// TIA Portal V20 export
// export: Created 2026-07-16T12:58:51.2791599Z, ExportSetting WithDefaults, DisplayName Totally Integrated Automation Portal, DisplayVersion V20 Update 5, DisplayName TIA Portal Openness, DisplayVersion V20 Update 4, DisplayName TIA Portal Version Control Interface, DisplayVersion V20 Update 5, DisplayName SINAMICS Startdrive Advanced, DisplayVersion V20, DisplayName SINAMICS DCC, DisplayVersion V20, DisplayName SINAMICS Startdrive G130, G150, S120, S150, SINAMICS MV, G220, S200, S210, DisplayVersion V20, DisplayName SINAMICS Startdrive G110M, G120, G120C, G120D, G120P, G115D, DisplayVersion V20, DisplayName STEP 7 Professional, DisplayVersion V20 Update 5, DisplayName STEP 7 Safety, DisplayVersion V20 Update 2, DisplayName WinCC Basic/Comfort/Advanced, DisplayVersion V20 Update 5, DisplayName WinCC Unified, DisplayVersion V20 Update 5
FUNCTION_BLOCK "FB_PusherControl"   // FB3, LAD
TITLE = Pusher Control
{ S7_Optimized_Access := 'TRUE' }
VERSION : 0.1
// Pusher ram sequencing (C-118-C-125). Step legend (C-120): 0=Parked (idle/home, ram fully retracted, no motion) - 10=DriveToEndTravel (forward stroke in progress) - 20=Hold (paused at full travel, brief settle before retracting) - 30=Retract (returning to home; also the recovery/abort target from any bad state). Mode legend: 0=Off (finish a retract already in progress, then park; no new cycle starts) - 1=Auto (hopper-high-level starts a cycle) - 2=Manual (operator button/jog starts a cycle).
// stored: AutoNumber true, IsIECCheckEnabled false, IsRetainMemResEnabled false, MemoryReserve 100, SetENOAutomatically false, UDAEnableTagReadback false
   VAR RETAIN
      IO { S7_SetPoint := 'True'} : "UDT_PusherIO";   // Caller-visible interface (C-115) - FC_ControlMain writes Mode/HopperHighLevel/limits/tunables in, reads Extend/Retract/RunPowerPack/fault bits out. See the block header for the Step/Mode value legend.
   END_VAR
   VAR
      EndTravelTimeoutMS : DInt;
      ParkedTimeoutMS : DInt;
      EndTravelHoldTimeMS : DInt;
      PumpRunOnTimeMS : DInt;
      JogWarningTimeMS : DInt;
      PressureTripConfirmTimeMS : DInt;
      PressureClearResumeDelayMS : DInt;
      PressureConfirmTimer { S7_SetPoint := 'True'} : TON_TIME;
      PressureClearTimer { S7_SetPoint := 'True'} : TON_TIME;
      PressureHold : Bool;   // Latched jam hold, not a fault (C-123) - see the Pressure Detection network. Freezes ExtendDemand while set; clears itself once pressure has genuinely stayed clear for PressureClearResumeDelay.
      PressureConfirmEdge : Bool;
      PressureConfirmEdgeMem : Bool;
      PressureTripCount : Int;   // Confirmed jams this cycle - reset each cycle start, not time-windowed. Compared against IO.PressureTripCountThreshold to raise Blocked.
      EndTravelTimer { S7_SetPoint := 'True'} : TON_TIME;
      HoldTimer { S7_SetPoint := 'True'} : TON_TIME;
      ParkedTimer { S7_SetPoint := 'True'} : TON_TIME;
      JogPreStartTimer { S7_SetPoint := 'True'} : TON_TIME;
      ExtendDemand : Bool;
      RetractDemand : Bool;
      PumpDemand : Bool;   // ExtendDemand OR RetractDemand - the pump's own immediate (non-run-on) demand signal.
      PumpEverDemanded : Bool;   // Cold-start guard for the pump run-on off-delay below - see that network's own comment.
      PumpRunOnTimer { S7_SetPoint := 'True'} : TON_TIME;
   END_VAR
   VAR_TEMP
      "Time" : Real;
   END_VAR
BEGIN

REGION Network 1: Enable
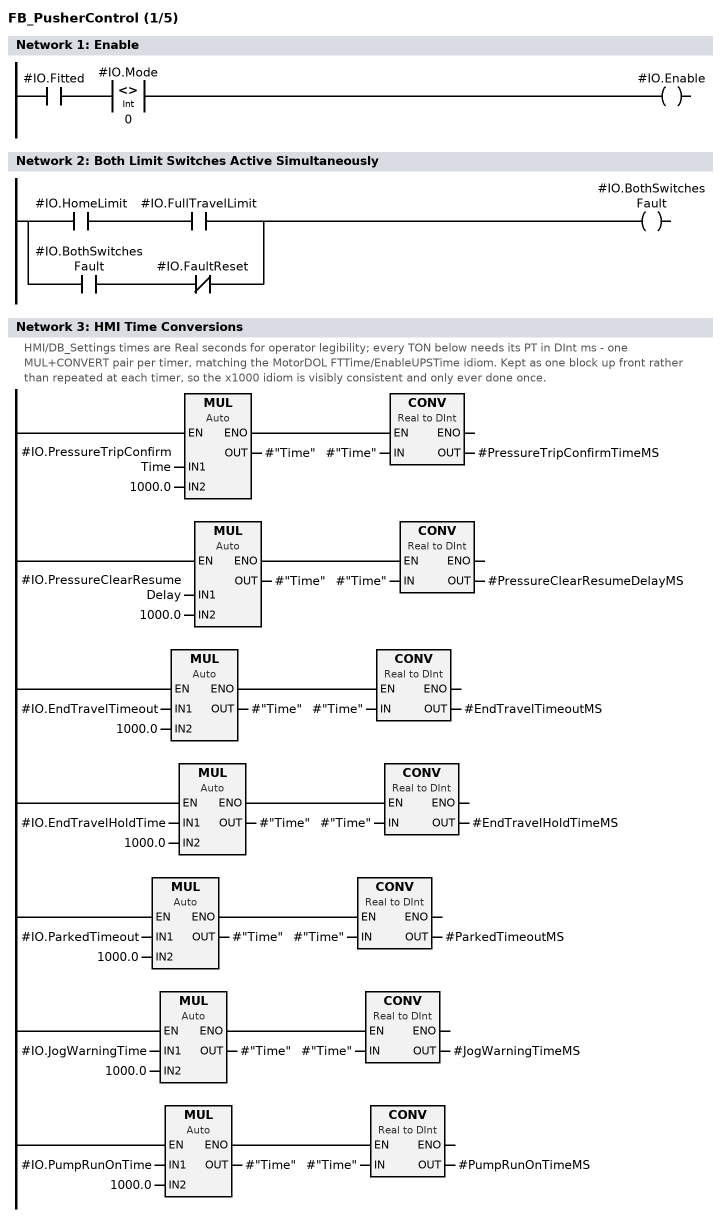
   RUNG wire#powerrail
      Contact( #IO.Fitted )
      { S7_Templates := "SrcType := Int" } NE_Contact(in1 := #IO.Mode, in2 := 0)
      Coil( #IO.Enable )
   END_RUNG
   // the same network as SCL:
   #IO.Enable := #IO.Fitted AND (#IO.Mode <> 0);
END_REGION

REGION Network 2: Both Limit Switches Active Simultaneously
   RUNG wire#powerrail
      Contact( #IO.HomeLimit )
      Contact( #IO.FullTravelLimit )
      wire#w1
      Coil( #IO.BothSwitchesFault )
   END_RUNG
   RUNG wire#powerrail
      Contact( #IO.BothSwitchesFault )
      I_Contact( #IO.FaultReset )
   END_RUNG wire#w1
   // the same network as SCL:
   #IO.BothSwitchesFault := (#IO.HomeLimit AND #IO.FullTravelLimit) OR (#IO.BothSwitchesFault AND NOT #IO.FaultReset);
END_REGION

REGION Network 3: HMI Time Conversions
   // HMI/DB_Settings times are Real seconds for operator legibility; every TON below needs its PT in DInt ms - one MUL+CONVERT pair per timer, matching the MotorDOL FTTime/EnableUPSTime idiom. Kept as one block up front rather than repeated at each timer, so the x1000 idiom is visibly consistent and only ever done once.
   RUNG wire#powerrail
      Mul(in1 := #IO.PressureTripConfirmTime, in2 := 1000.0, out => #"Time")
      { S7_Templates := "[SrcType := Real, DestType := DInt]" } Convert(in := #"Time", out => #PressureTripConfirmTimeMS)
   END_RUNG
   RUNG wire#powerrail
      Mul(in1 := #IO.PressureClearResumeDelay, in2 := 1000.0, out => #"Time")
      { S7_Templates := "[SrcType := Real, DestType := DInt]" } Convert(in := #"Time", out => #PressureClearResumeDelayMS)
   END_RUNG
   RUNG wire#powerrail
      Mul(in1 := #IO.EndTravelTimeout, in2 := 1000.0, out => #"Time")
      { S7_Templates := "[SrcType := Real, DestType := DInt]" } Convert(in := #"Time", out => #EndTravelTimeoutMS)
   END_RUNG
   RUNG wire#powerrail
      Mul(in1 := #IO.EndTravelHoldTime, in2 := 1000.0, out => #"Time")
      { S7_Templates := "[SrcType := Real, DestType := DInt]" } Convert(in := #"Time", out => #EndTravelHoldTimeMS)
   END_RUNG
   RUNG wire#powerrail
      Mul(in1 := #IO.ParkedTimeout, in2 := 1000.0, out => #"Time")
      { S7_Templates := "[SrcType := Real, DestType := DInt]" } Convert(in := #"Time", out => #ParkedTimeoutMS)
   END_RUNG
   RUNG wire#powerrail
      Mul(in1 := #IO.JogWarningTime, in2 := 1000.0, out => #"Time")
      { S7_Templates := "[SrcType := Real, DestType := DInt]" } Convert(in := #"Time", out => #JogWarningTimeMS)
   END_RUNG
   RUNG wire#powerrail
      Mul(in1 := #IO.PumpRunOnTime, in2 := 1000.0, out => #"Time")
      { S7_Templates := "[SrcType := Real, DestType := DInt]" } Convert(in := #"Time", out => #PumpRunOnTimeMS)
   END_RUNG
   // the same network as SCL:
   #"Time" := #IO.PressureTripConfirmTime * 1000.0;
   #PressureTripConfirmTimeMS := REAL_TO_DINT(#"Time");
   #"Time" := #IO.PressureClearResumeDelay * 1000.0;
   #PressureClearResumeDelayMS := REAL_TO_DINT(#"Time");
   #"Time" := #IO.EndTravelTimeout * 1000.0;
   #EndTravelTimeoutMS := REAL_TO_DINT(#"Time");
   #"Time" := #IO.EndTravelHoldTime * 1000.0;
   #EndTravelHoldTimeMS := REAL_TO_DINT(#"Time");
   #"Time" := #IO.ParkedTimeout * 1000.0;
   #ParkedTimeoutMS := REAL_TO_DINT(#"Time");
   #"Time" := #IO.JogWarningTime * 1000.0;
   #JogWarningTimeMS := REAL_TO_DINT(#"Time");
   #"Time" := #IO.PumpRunOnTime * 1000.0;
   #PumpRunOnTimeMS := REAL_TO_DINT(#"Time");
END_REGION

REGION Network 4: Pressure Trip Detection, Hold, And Counting
   // One function, one network: a trip must be debounced (PressureConfirmTimer) before it counts - momentary pressure spikes aren't a real jam. Hold latches through a confirmed trip and only releases once pressure has genuinely cleared for PressureClearResumeDelay, so a bouncing switch can't re-trigger the count on every scan. Count resets each cycle start (Step 0-to-10 launch condition), not on a rolling time window.
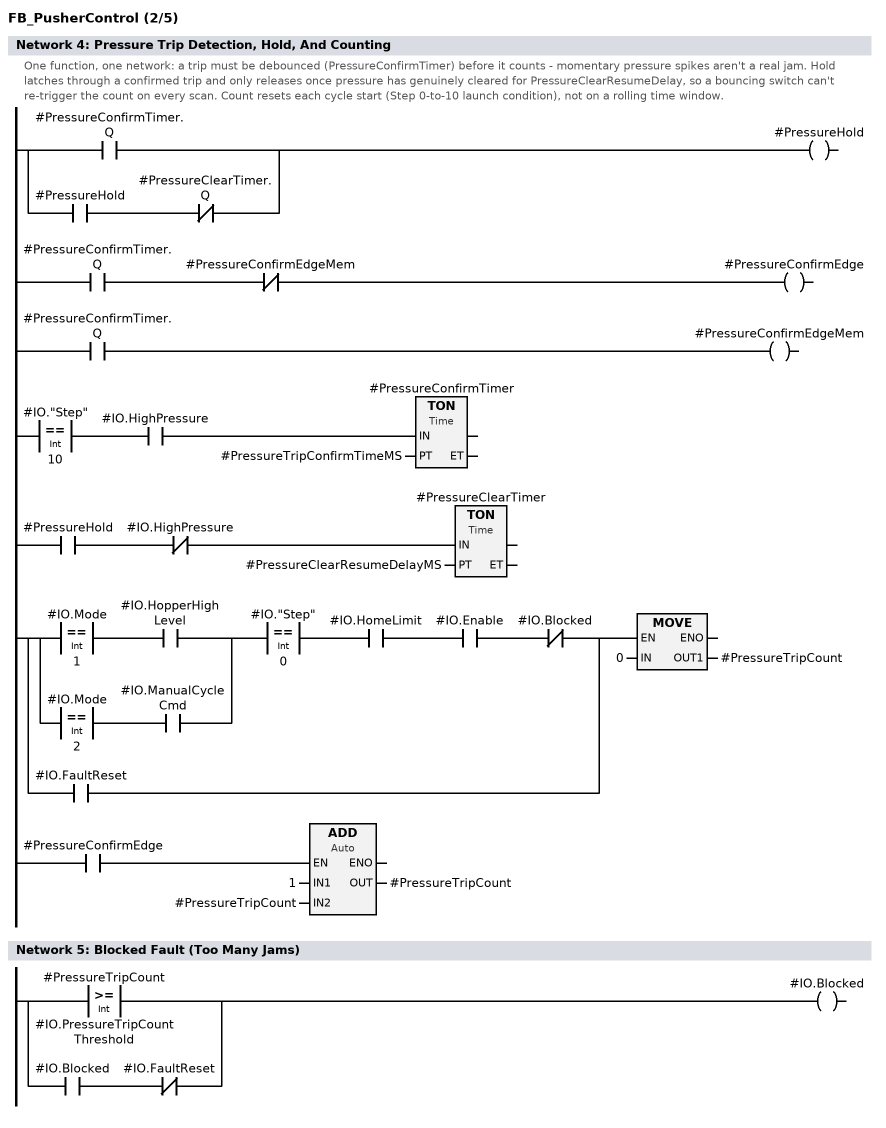
   RUNG wire#powerrail
      Contact( #PressureConfirmTimer.Q )
      wire#w1
      Coil( #PressureHold )
   END_RUNG
   RUNG wire#powerrail
      Contact( #PressureHold )
      I_Contact( #PressureClearTimer.Q )
   END_RUNG wire#w1
   RUNG wire#powerrail
      Contact( #PressureConfirmTimer.Q )
      I_Contact( #PressureConfirmEdgeMem )
      Coil( #PressureConfirmEdge )
   END_RUNG
   RUNG wire#powerrail
      Contact( #PressureConfirmTimer.Q )
      Coil( #PressureConfirmEdgeMem )
   END_RUNG
   RUNG wire#powerrail
      { S7_Templates := "SrcType := Int" } EQ_Contact(in1 := #IO."Step", in2 := 10)
      Contact( #IO.HighPressure )
      { S7_Templates := "time_type := Time" } #PressureConfirmTimer.TON(pt := #PressureTripConfirmTimeMS, et =>)
   END_RUNG
   RUNG wire#powerrail
      Contact( #PressureHold )
      I_Contact( #IO.HighPressure )
      { S7_Templates := "time_type := Time" } #PressureClearTimer.TON(pt := #PressureClearResumeDelayMS, et =>)
   END_RUNG
   RUNG wire#powerrail
      { S7_Templates := "SrcType := Int" } EQ_Contact(in1 := #IO.Mode, in2 := 1)
      Contact( #IO.HopperHighLevel )
      wire#w2
      { S7_Templates := "SrcType := Int" } EQ_Contact(in1 := #IO."Step", in2 := 0)
      Contact( #IO.HomeLimit )
      Contact( #IO.Enable )
      I_Contact( #IO.Blocked )
      wire#w3
      Move(in := 0, out1 => #PressureTripCount)
   END_RUNG
   RUNG wire#powerrail
      { S7_Templates := "SrcType := Int" } EQ_Contact(in1 := #IO.Mode, in2 := 2)
      Contact( #IO.ManualCycleCmd )
   END_RUNG wire#w2
   RUNG wire#powerrail
      Contact( #IO.FaultReset )
   END_RUNG wire#w3
   RUNG wire#powerrail
      Contact( #PressureConfirmEdge )
      Add(in1 := 1, in2 := #PressureTripCount, out => #PressureTripCount)
   END_RUNG
   // the same network as SCL:
   #PressureHold := #PressureConfirmTimer.Q OR (#PressureHold AND NOT #PressureClearTimer.Q);
   #PressureConfirmEdge := #PressureConfirmTimer.Q AND NOT #PressureConfirmEdgeMem;
   #PressureConfirmEdgeMem := #PressureConfirmTimer.Q;
   #PressureConfirmTimer(IN := (#IO."Step" = 10) AND #IO.HighPressure, PT := #PressureTripConfirmTimeMS);   // TON
   #PressureClearTimer(IN := #PressureHold AND NOT #IO.HighPressure, PT := #PressureClearResumeDelayMS);   // TON
   IF ((((#IO.Mode = 1) AND #IO.HopperHighLevel) OR ((#IO.Mode = 2) AND #IO.ManualCycleCmd)) AND (#IO."Step" = 0) AND #IO.HomeLimit AND #IO.Enable AND NOT #IO.Blocked) OR #IO.FaultReset THEN
       #PressureTripCount := 0;
   END_IF;
   IF #PressureConfirmEdge THEN #PressureTripCount := 1 + #PressureTripCount; END_IF;
END_REGION

REGION Network 5: Blocked Fault (Too Many Jams)
   RUNG wire#powerrail
      { S7_Templates := "SrcType := Int" } GE_Contact(in1 := #PressureTripCount, in2 := #IO.PressureTripCountThreshold)
      wire#w1
      Coil( #IO.Blocked )
   END_RUNG
   RUNG wire#powerrail
      Contact( #IO.Blocked )
      I_Contact( #IO.FaultReset )
   END_RUNG wire#w1
   // the same network as SCL:
   #IO.Blocked := (#PressureTripCount >= #IO.PressureTripCountThreshold) OR (#IO.Blocked AND NOT #IO.FaultReset);
END_REGION

REGION Network 6: Step 0 (Parked) - Transitions
   // Not-at-home while idle (power-up mid-stroke, or a cycle that ended without reaching HomeLimit) drives straight to Retract (30) to re-establish home before any new cycle is accepted - never straight back into a forward stroke from an unknown position. Suppressed during an active jog command so jogging isn't fought by an auto-retract.
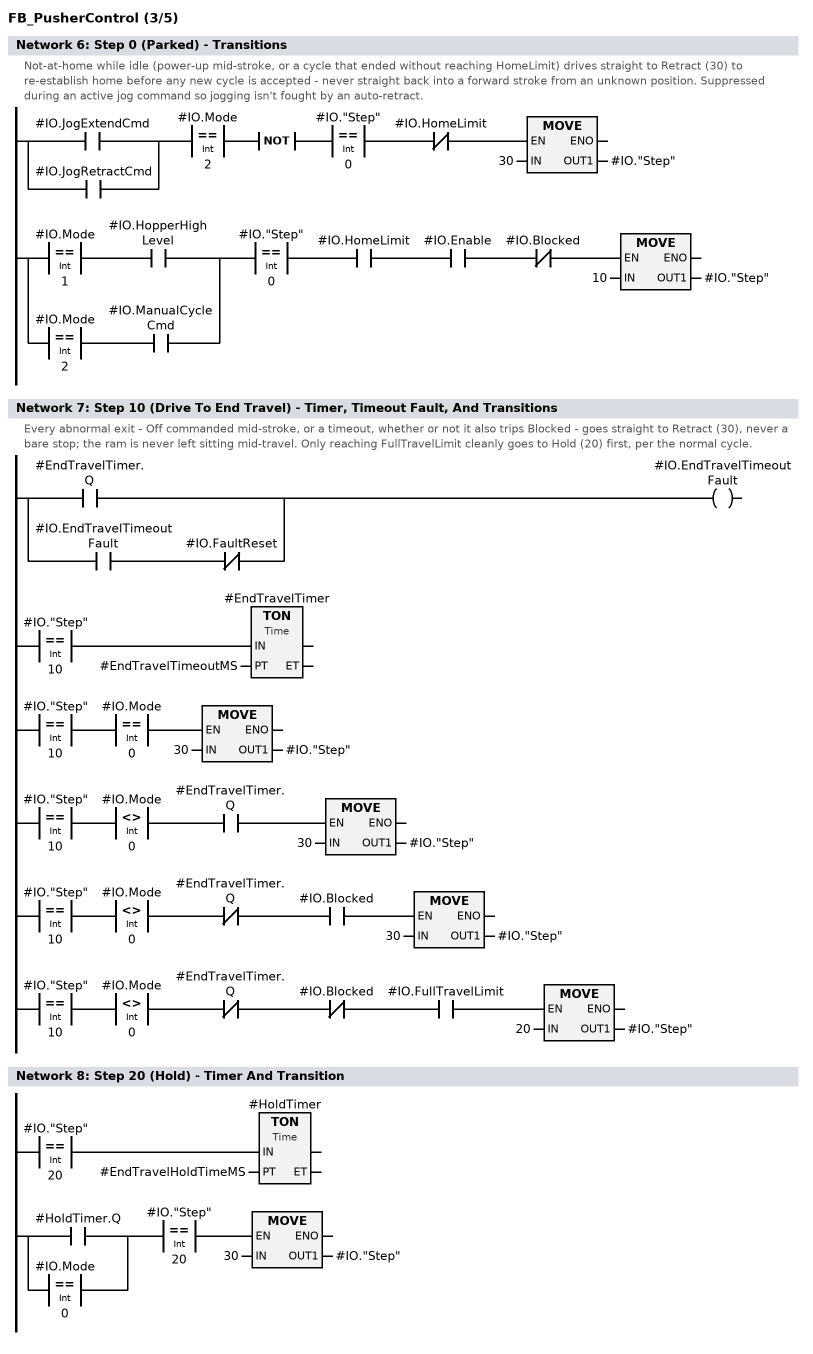
   RUNG wire#powerrail
      Contact( #IO.JogExtendCmd )
      wire#w1
      { S7_Templates := "SrcType := Int" } EQ_Contact(in1 := #IO.Mode, in2 := 2)
      Not()
      { S7_Templates := "SrcType := Int" } EQ_Contact(in1 := #IO."Step", in2 := 0)
      I_Contact( #IO.HomeLimit )
      Move(in := 30, out1 => #IO."Step")
   END_RUNG
   RUNG wire#powerrail
      Contact( #IO.JogRetractCmd )
   END_RUNG wire#w1
   RUNG wire#powerrail
      { S7_Templates := "SrcType := Int" } EQ_Contact(in1 := #IO.Mode, in2 := 1)
      Contact( #IO.HopperHighLevel )
      wire#w2
      { S7_Templates := "SrcType := Int" } EQ_Contact(in1 := #IO."Step", in2 := 0)
      Contact( #IO.HomeLimit )
      Contact( #IO.Enable )
      I_Contact( #IO.Blocked )
      Move(in := 10, out1 => #IO."Step")
   END_RUNG
   RUNG wire#powerrail
      { S7_Templates := "SrcType := Int" } EQ_Contact(in1 := #IO.Mode, in2 := 2)
      Contact( #IO.ManualCycleCmd )
   END_RUNG wire#w2
   // the same network as SCL:
   IF NOT ((#IO.JogExtendCmd OR #IO.JogRetractCmd) AND (#IO.Mode = 2)) AND (#IO."Step" = 0) AND NOT #IO.HomeLimit THEN
       #IO."Step" := 30;
   END_IF;
   IF (((#IO.Mode = 1) AND #IO.HopperHighLevel) OR ((#IO.Mode = 2) AND #IO.ManualCycleCmd)) AND (#IO."Step" = 0) AND #IO.HomeLimit AND #IO.Enable AND NOT #IO.Blocked THEN
       #IO."Step" := 10;
   END_IF;
END_REGION

REGION Network 7: Step 10 (Drive To End Travel) - Timer, Timeout Fault, And Transitions
   // Every abnormal exit - Off commanded mid-stroke, or a timeout, whether or not it also trips Blocked - goes straight to Retract (30), never a bare stop; the ram is never left sitting mid-travel. Only reaching FullTravelLimit cleanly goes to Hold (20) first, per the normal cycle.
   RUNG wire#powerrail
      Contact( #EndTravelTimer.Q )
      wire#w1
      Coil( #IO.EndTravelTimeoutFault )
   END_RUNG
   RUNG wire#powerrail
      Contact( #IO.EndTravelTimeoutFault )
      I_Contact( #IO.FaultReset )
   END_RUNG wire#w1
   RUNG wire#powerrail
      { S7_Templates := "SrcType := Int" } EQ_Contact(in1 := #IO."Step", in2 := 10)
      { S7_Templates := "time_type := Time" } #EndTravelTimer.TON(pt := #EndTravelTimeoutMS, et =>)
   END_RUNG
   RUNG wire#powerrail
      { S7_Templates := "SrcType := Int" } EQ_Contact(in1 := #IO."Step", in2 := 10)
      { S7_Templates := "SrcType := Int" } EQ_Contact(in1 := #IO.Mode, in2 := 0)
      Move(in := 30, out1 => #IO."Step")
   END_RUNG
   RUNG wire#powerrail
      { S7_Templates := "SrcType := Int" } EQ_Contact(in1 := #IO."Step", in2 := 10)
      { S7_Templates := "SrcType := Int" } NE_Contact(in1 := #IO.Mode, in2 := 0)
      Contact( #EndTravelTimer.Q )
      Move(in := 30, out1 => #IO."Step")
   END_RUNG
   RUNG wire#powerrail
      { S7_Templates := "SrcType := Int" } EQ_Contact(in1 := #IO."Step", in2 := 10)
      { S7_Templates := "SrcType := Int" } NE_Contact(in1 := #IO.Mode, in2 := 0)
      I_Contact( #EndTravelTimer.Q )
      Contact( #IO.Blocked )
      Move(in := 30, out1 => #IO."Step")
   END_RUNG
   RUNG wire#powerrail
      { S7_Templates := "SrcType := Int" } EQ_Contact(in1 := #IO."Step", in2 := 10)
      { S7_Templates := "SrcType := Int" } NE_Contact(in1 := #IO.Mode, in2 := 0)
      I_Contact( #EndTravelTimer.Q )
      I_Contact( #IO.Blocked )
      Contact( #IO.FullTravelLimit )
      Move(in := 20, out1 => #IO."Step")
   END_RUNG
   // the same network as SCL:
   #IO.EndTravelTimeoutFault := #EndTravelTimer.Q OR (#IO.EndTravelTimeoutFault AND NOT #IO.FaultReset);
   #EndTravelTimer(IN := #IO."Step" = 10, PT := #EndTravelTimeoutMS);   // TON
   IF (#IO."Step" = 10) AND (#IO.Mode = 0) THEN #IO."Step" := 30; END_IF;
   IF (#IO."Step" = 10) AND (#IO.Mode <> 0) AND #EndTravelTimer.Q THEN #IO."Step" := 30; END_IF;
   IF (#IO."Step" = 10) AND (#IO.Mode <> 0) AND NOT #EndTravelTimer.Q AND #IO.Blocked THEN
       #IO."Step" := 30;
   END_IF;
   IF (#IO."Step" = 10) AND (#IO.Mode <> 0) AND NOT #EndTravelTimer.Q AND NOT #IO.Blocked AND #IO.FullTravelLimit THEN
       #IO."Step" := 20;
   END_IF;
END_REGION

REGION Network 8: Step 20 (Hold) - Timer And Transition
   RUNG wire#powerrail
      { S7_Templates := "SrcType := Int" } EQ_Contact(in1 := #IO."Step", in2 := 20)
      { S7_Templates := "time_type := Time" } #HoldTimer.TON(pt := #EndTravelHoldTimeMS, et =>)
   END_RUNG
   RUNG wire#powerrail
      Contact( #HoldTimer.Q )
      wire#w1
      { S7_Templates := "SrcType := Int" } EQ_Contact(in1 := #IO."Step", in2 := 20)
      Move(in := 30, out1 => #IO."Step")
   END_RUNG
   RUNG wire#powerrail
      { S7_Templates := "SrcType := Int" } EQ_Contact(in1 := #IO.Mode, in2 := 0)
   END_RUNG wire#w1
   // the same network as SCL:
   #HoldTimer(IN := #IO."Step" = 20, PT := #EndTravelHoldTimeMS);   // TON
   IF (#HoldTimer.Q OR (#IO.Mode = 0)) AND (#IO."Step" = 20) THEN #IO."Step" := 30; END_IF;
END_REGION

REGION Network 9: Step 30 (Retract) - Timer, Timeout Fault, And Transition
   // ParkedTimer's own Q only feeds the timeout fault, not a transition - if genuinely stuck retracting there's no safer step to force (unlike Step 10, nothing here can be aborted into); alarm-only by design, awaiting a human.
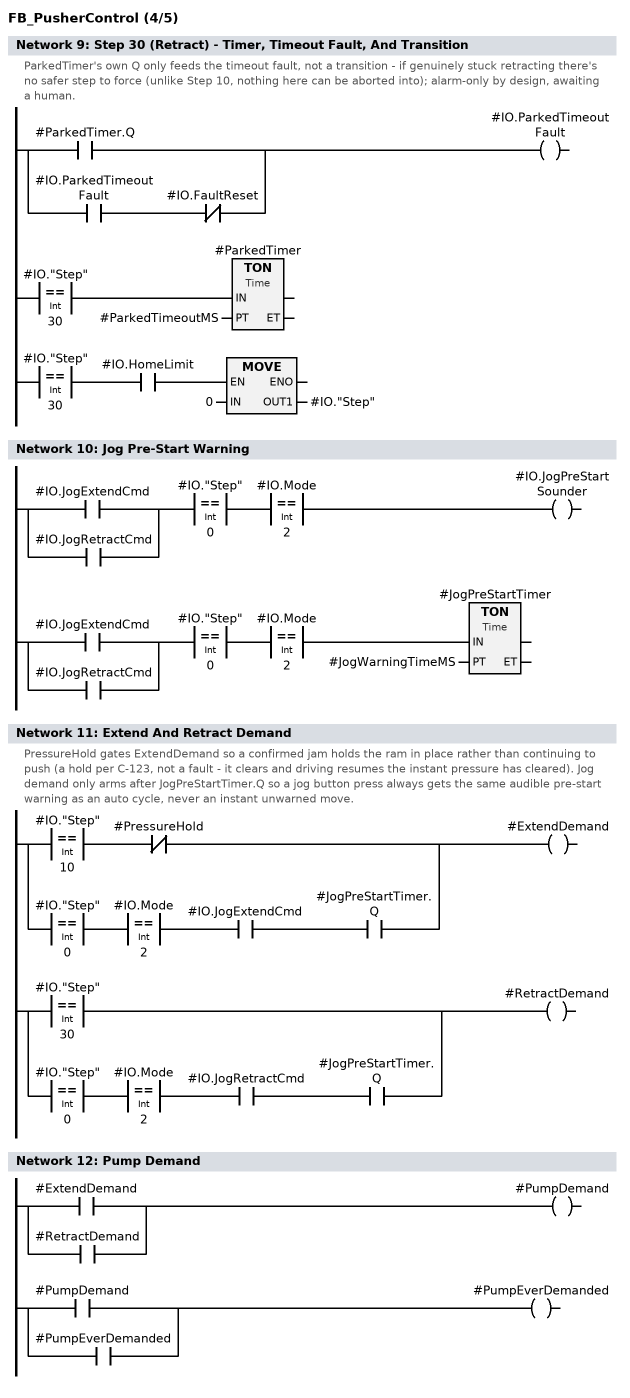
   RUNG wire#powerrail
      Contact( #ParkedTimer.Q )
      wire#w1
      Coil( #IO.ParkedTimeoutFault )
   END_RUNG
   RUNG wire#powerrail
      Contact( #IO.ParkedTimeoutFault )
      I_Contact( #IO.FaultReset )
   END_RUNG wire#w1
   RUNG wire#powerrail
      { S7_Templates := "SrcType := Int" } EQ_Contact(in1 := #IO."Step", in2 := 30)
      { S7_Templates := "time_type := Time" } #ParkedTimer.TON(pt := #ParkedTimeoutMS, et =>)
   END_RUNG
   RUNG wire#powerrail
      { S7_Templates := "SrcType := Int" } EQ_Contact(in1 := #IO."Step", in2 := 30)
      Contact( #IO.HomeLimit )
      Move(in := 0, out1 => #IO."Step")
   END_RUNG
   // the same network as SCL:
   #IO.ParkedTimeoutFault := #ParkedTimer.Q OR (#IO.ParkedTimeoutFault AND NOT #IO.FaultReset);
   #ParkedTimer(IN := #IO."Step" = 30, PT := #ParkedTimeoutMS);   // TON
   IF (#IO."Step" = 30) AND #IO.HomeLimit THEN #IO."Step" := 0; END_IF;
END_REGION

REGION Network 10: Jog Pre-Start Warning
   RUNG wire#powerrail
      Contact( #IO.JogExtendCmd )
      wire#w1
      { S7_Templates := "SrcType := Int" } EQ_Contact(in1 := #IO."Step", in2 := 0)
      { S7_Templates := "SrcType := Int" } EQ_Contact(in1 := #IO.Mode, in2 := 2)
      Coil( #IO.JogPreStartSounder )
   END_RUNG
   RUNG wire#powerrail
      Contact( #IO.JogRetractCmd )
   END_RUNG wire#w1
   RUNG wire#powerrail
      Contact( #IO.JogExtendCmd )
      wire#w2
      { S7_Templates := "SrcType := Int" } EQ_Contact(in1 := #IO."Step", in2 := 0)
      { S7_Templates := "SrcType := Int" } EQ_Contact(in1 := #IO.Mode, in2 := 2)
      { S7_Templates := "time_type := Time" } #JogPreStartTimer.TON(pt := #JogWarningTimeMS, et =>)
   END_RUNG
   RUNG wire#powerrail
      Contact( #IO.JogRetractCmd )
   END_RUNG wire#w2
   // the same network as SCL:
   #IO.JogPreStartSounder := (#IO.JogExtendCmd OR #IO.JogRetractCmd) AND (#IO."Step" = 0) AND (#IO.Mode = 2);
   #JogPreStartTimer(IN := (#IO.JogExtendCmd OR #IO.JogRetractCmd) AND (#IO."Step" = 0) AND (#IO.Mode = 2),   // TON
                     PT := #JogWarningTimeMS);
END_REGION

REGION Network 11: Extend And Retract Demand
   // PressureHold gates ExtendDemand so a confirmed jam holds the ram in place rather than continuing to push (a hold per C-123, not a fault - it clears and driving resumes the instant pressure has cleared). Jog demand only arms after JogPreStartTimer.Q so a jog button press always gets the same audible pre-start warning as an auto cycle, never an instant unwarned move.
   RUNG wire#powerrail
      { S7_Templates := "SrcType := Int" } EQ_Contact(in1 := #IO."Step", in2 := 10)
      I_Contact( #PressureHold )
      wire#w1
      Coil( #ExtendDemand )
   END_RUNG
   RUNG wire#powerrail
      { S7_Templates := "SrcType := Int" } EQ_Contact(in1 := #IO."Step", in2 := 0)
      { S7_Templates := "SrcType := Int" } EQ_Contact(in1 := #IO.Mode, in2 := 2)
      Contact( #IO.JogExtendCmd )
      Contact( #JogPreStartTimer.Q )
   END_RUNG wire#w1
   RUNG wire#powerrail
      { S7_Templates := "SrcType := Int" } EQ_Contact(in1 := #IO."Step", in2 := 30)
      wire#w2
      Coil( #RetractDemand )
   END_RUNG
   RUNG wire#powerrail
      { S7_Templates := "SrcType := Int" } EQ_Contact(in1 := #IO."Step", in2 := 0)
      { S7_Templates := "SrcType := Int" } EQ_Contact(in1 := #IO.Mode, in2 := 2)
      Contact( #IO.JogRetractCmd )
      Contact( #JogPreStartTimer.Q )
   END_RUNG wire#w2
   // the same network as SCL:
   #ExtendDemand := ((#IO."Step" = 10) AND NOT #PressureHold) OR ((#IO."Step" = 0) AND (#IO.Mode = 2) AND #IO.JogExtendCmd AND #JogPreStartTimer.Q);
   #RetractDemand := (#IO."Step" = 30) OR ((#IO."Step" = 0) AND (#IO.Mode = 2) AND #IO.JogRetractCmd AND #JogPreStartTimer.Q);
END_REGION

REGION Network 12: Pump Demand
   RUNG wire#powerrail
      Contact( #ExtendDemand )
      wire#w1
      Coil( #PumpDemand )
   END_RUNG
   RUNG wire#powerrail
      Contact( #RetractDemand )
   END_RUNG wire#w1
   RUNG wire#powerrail
      Contact( #PumpDemand )
      wire#w2
      Coil( #PumpEverDemanded )
   END_RUNG
   RUNG wire#powerrail
      Contact( #PumpEverDemanded )
   END_RUNG wire#w2
   // the same network as SCL:
   #PumpDemand := #ExtendDemand OR #RetractDemand;
   #PumpEverDemanded := #PumpDemand OR #PumpEverDemanded;
END_REGION

REGION Network 13: Pump Run-On Timer And Output Commands
   // Off-delay built from TON+inversion, not TOF/TONR (C-406). PumpEverDemanded guards a cold-start gap: on power-up PumpDemand and the timer's Q are both initially false, which would read as 'run-on already elapsed' and skip straight to no-run. RunPowerPack stays on through the run-on tail even after demand drops, but the Extend/Retract solenoids are not - they only ever follow live demand, gated by PowerPackRunningFB so the ram can't be commanded before the pump has confirmed running.
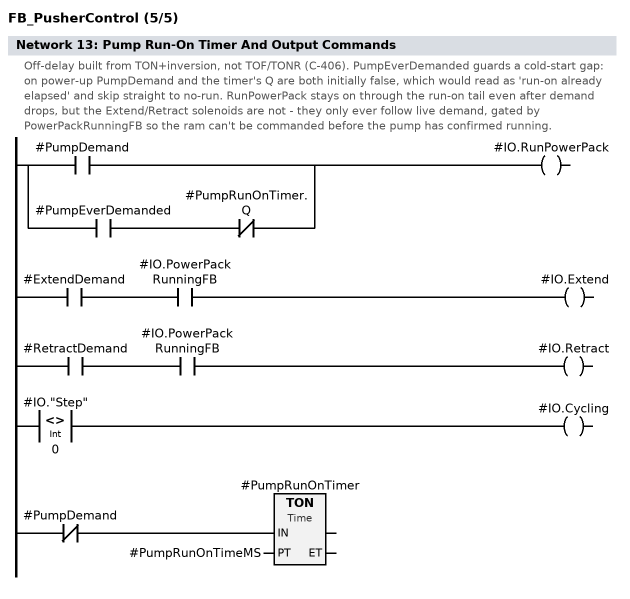
   RUNG wire#powerrail
      Contact( #PumpDemand )
      wire#w1
      Coil( #IO.RunPowerPack )
   END_RUNG
   RUNG wire#powerrail
      Contact( #PumpEverDemanded )
      I_Contact( #PumpRunOnTimer.Q )
   END_RUNG wire#w1
   RUNG wire#powerrail
      Contact( #ExtendDemand )
      Contact( #IO.PowerPackRunningFB )
      Coil( #IO.Extend )
   END_RUNG
   RUNG wire#powerrail
      Contact( #RetractDemand )
      Contact( #IO.PowerPackRunningFB )
      Coil( #IO.Retract )
   END_RUNG
   RUNG wire#powerrail
      { S7_Templates := "SrcType := Int" } NE_Contact(in1 := #IO."Step", in2 := 0)
      Coil( #IO.Cycling )
   END_RUNG
   RUNG wire#powerrail
      I_Contact( #PumpDemand )
      { S7_Templates := "time_type := Time" } #PumpRunOnTimer.TON(pt := #PumpRunOnTimeMS, et =>)
   END_RUNG
   // the same network as SCL:
   #IO.RunPowerPack := #PumpDemand OR (#PumpEverDemanded AND NOT #PumpRunOnTimer.Q);
   #IO.Extend := #ExtendDemand AND #IO.PowerPackRunningFB;
   #IO.Retract := #RetractDemand AND #IO.PowerPackRunningFB;
   #IO.Cycling := #IO."Step" <> 0;
   #PumpRunOnTimer(IN := NOT #PumpDemand, PT := #PumpRunOnTimeMS);   // TON
END_REGION
END_FUNCTION_BLOCK
